// TIA Portal V20 export
// export: Created 2026-07-14T14:10:15.7260647Z, ExportSetting WithDefaults, DisplayName Totally Integrated Automation Portal, DisplayVersion V20 Update 5, DisplayName TIA Portal Openness, DisplayVersion V20 Update 4, DisplayName TIA Portal Version Control Interface, DisplayVersion V20 Update 5, DisplayName SINAMICS Startdrive Advanced, DisplayVersion V20, DisplayName SINAMICS DCC, DisplayVersion V20, DisplayName SINAMICS Startdrive G130, G150, S120, S150, SINAMICS MV, G220, S200, S210, DisplayVersion V20, DisplayName SINAMICS Startdrive G110M, G120, G120C, G120D, G120P, G115D, DisplayVersion V20, DisplayName STEP 7 Professional, DisplayVersion V20 Update 5, DisplayName STEP 7 Safety, DisplayVersion V20 Update 2, DisplayName WinCC Basic/Comfort/Advanced, DisplayVersion V20 Update 5, DisplayName WinCC Unified, DisplayVersion V20 Update 5
FUNCTION "SignalConditioning" : Void   // FC21, LAD
{ S7_Optimized_Access := 'TRUE' }
VERSION : 0.1
// Arithmetic/box-instruction reference examples (Mul/Convert/Sub/Div/Abs/Swap)
// stored: AutoNumber true, IsIECCheckEnabled false, SetENOAutomatically false, UDAEnableTagReadback false
   VAR_TEMP
      SpeedRawA : Real;
      ScaleFactor : Real;
      SpeedScaled : Real;
      SpeedScaledSource : Real;
      SpeedConverted : DInt;
      Enable : Bool;
      Level : Int;
      MinuendA : Int;
      SubtrahendA : Int;
      Difference : Int;
      DividendB : Int;
      DivisorB : Int;
      Quotient : Int;
      GateBit : Bool;
      SignedValue : Real;
      AbsValue : Real;
      ControlWord : Word;
      SwappedWord : Word;
   END_VAR
BEGIN

REGION Network 1: Speed scaling (Mul/Convert)
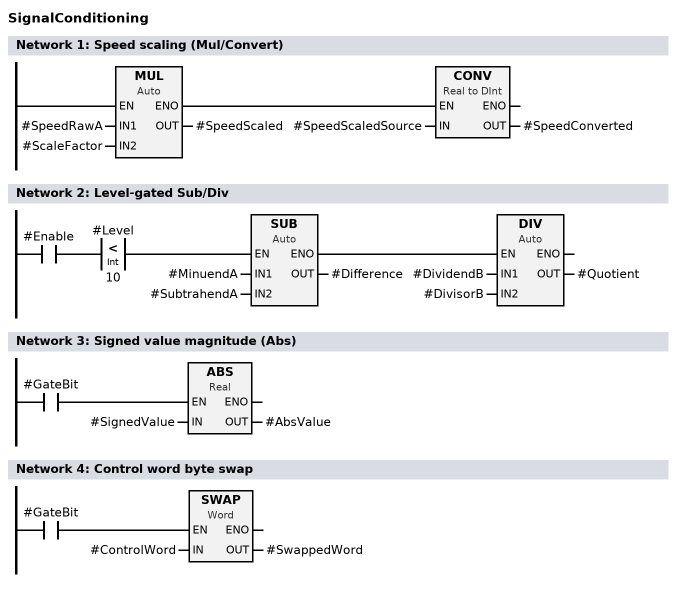
   RUNG wire#powerrail
      Mul(in1 := #SpeedRawA, in2 := #ScaleFactor, out => #SpeedScaled)
      { S7_Templates := "[SrcType := Real, DestType := DInt]" } Convert(in := #SpeedScaledSource, out => #SpeedConverted)
   END_RUNG
   // the same network as SCL:
   #SpeedScaled := #SpeedRawA * #ScaleFactor;
   #SpeedConverted := REAL_TO_DINT(#SpeedScaledSource);
END_REGION

REGION Network 2: Level-gated Sub/Div
   RUNG wire#powerrail
      Contact( #Enable )
      { S7_Templates := "SrcType := Int" } LT_Contact(in1 := #Level, in2 := 10)
      Sub(in1 := #MinuendA, in2 := #SubtrahendA, out => #Difference)
      Div(in1 := #DividendB, in2 := #DivisorB, out => #Quotient)
   END_RUNG
   // the same network as SCL:
   IF #Enable AND (#Level < 10) THEN
       #Difference := #MinuendA - #SubtrahendA;
       #Quotient := #DividendB / #DivisorB;
   END_IF;
END_REGION

REGION Network 3: Signed value magnitude (Abs)
   RUNG wire#powerrail
      Contact( #GateBit )
      { S7_Templates := "SrcType := Real" } Abs(in := #SignedValue, out => #AbsValue)
   END_RUNG
   // the same network as SCL:
   IF #GateBit THEN #AbsValue := ABS(#SignedValue); END_IF;
END_REGION

REGION Network 4: Control word byte swap
   IF #GateBit THEN #SwappedWord := SWAP(#ControlWord); END_IF;
END_REGION
END_FUNCTION
